{attribute 'qualified_only'}
VAR_GLOBAL CONSTANT
	maxPairs : INT := 16;
	maxQueue : INT := 16;
END_VAR

(* stored: Version 1.1.0.1, ProductVersion 3.1.4024.11
   GVL GVL: Id {cd4bbf90-35e7-4ef6-9f55-dd1e548fe410} *)
